// TIA Portal V16 export
// export: Created 2022-04-14T22:37:40.7976404Z, ExportSetting WithDefaults, DisplayName Totally Integrated Automation Portal, DisplayVersion V16, DisplayName TIA Portal Version Control Interface, DisplayVersion V16, DisplayName TIA Portal Openness, DisplayVersion V16, DisplayName STEP 7 Professional, DisplayVersion V16, DisplayName STEP 7 Safety, DisplayVersion V16, DisplayName WinCC Professional, DisplayVersion V16
FUNCTION_BLOCK "01 Startup"   // FB1, LAD
{ S7_Optimized_Access := 'TRUE' }
VERSION : 0.1
// stored: AutoNumber true, IsIECCheckEnabled false, IsRetainMemResEnabled false, MemoryReserve 100, SetENOAutomatically false, UDAEnableTagReadback false
   VAR_TEMP   // added for the SCL form of the ladder/FBD networks
      _w1 : Bool;
   END_VAR
BEGIN

REGION Network 1: Run Mode
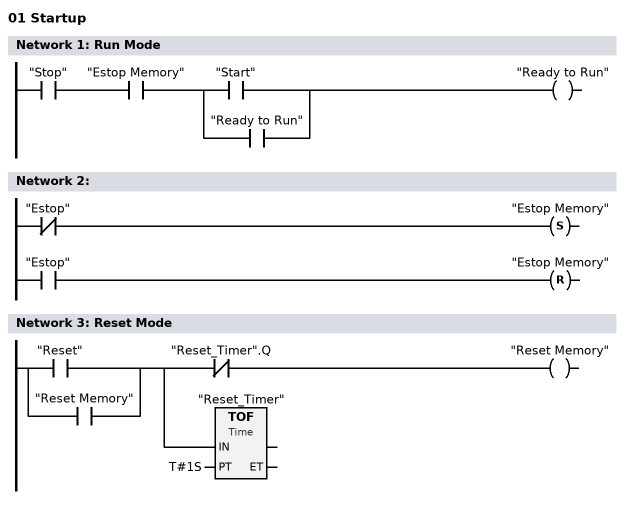
   RUNG wire#powerrail
      Contact( "Stop" )
      Contact( "Estop Memory" )
      wire#w1
      Contact( "Start" )
      wire#w2
      Coil( "Ready to Run" )
   END_RUNG
   RUNG wire#w1
      Contact( "Ready to Run" )
   END_RUNG wire#w2
   // the same network as SCL:
   "Ready to Run" := "Stop" AND "Estop Memory" AND ("Start" OR "Ready to Run");
END_REGION

REGION Network 2
   RUNG wire#powerrail
      I_Contact( "Estop" )
      S_Coil( "Estop Memory" )
   END_RUNG
   RUNG wire#powerrail
      Contact( "Estop" )
      R_Coil( "Estop Memory" )
   END_RUNG
   // the same network as SCL:
   IF NOT "Estop" THEN "Estop Memory" := TRUE; END_IF;
   IF "Estop" THEN "Estop Memory" := FALSE; END_IF;
END_REGION

REGION Network 3: Reset Mode
   RUNG wire#powerrail
      Contact( "Reset" )
      wire#w1
      I_Contact( "Reset_Timer".Q )
      Coil( "Reset Memory" )
   END_RUNG
   RUNG wire#powerrail
      Contact( "Reset Memory" )
   END_RUNG wire#w1
   RUNG wire#w1
      { S7_Templates := "time_type := Time" } "Reset_Timer".TOF(pt := T#1S, et =>)
   END_RUNG
   // the same network as SCL:
   #_w1 := "Reset" OR "Reset Memory";
   "Reset Memory" := #_w1 AND NOT "Reset_Timer".Q;
   "Reset_Timer".TOF(IN := #_w1, PT := T#1S);
END_REGION
END_FUNCTION_BLOCK
